TYPE ST_EP9224_in :
STRUCT
	stChannel : ARRAY [1..EP9224_NUM_CHANNELS] OF ST_EP9224_InputChannel;
	stInputDevice :ST_EP9224_InputDevice;
	bWcState : BOOL;
	nEcState : UINT;
END_STRUCT
END_TYPE

(* stored: Version 1.1.0.1, ProductVersion 3.1.4024.9
   DUT ST_EP9224_in: Id {226a3d55-dce3-4dcb-9cb7-bc45bfa31cef} *)
